FUNCTION_BLOCK fb_BusBrsEvent
VAR_INPUT
	 I_sID         			:STRING(10);     // Geräte-ID (z.B. '12345')
	 I_sInstID				:STRING(2) 	:=	'17';
	 I_sReceivedString		:STRING(255);	
	 I_bReset				:BOOL;
END_VAR
VAR_OUTPUT
	Q_lrBrs				:LREAL;
END_VAR
VAR	
	findStringTemp			:STRING;	(* Wird für TMP/ BRS/ RHD verwendet *)

	sBrs1					:STRING;
	sBrs2					:STRING;
	
END_VAR

findStringTemp	:= CONCAT(I_sID,'.');
findStringTemp	:= CONCAT(findStringTemp,'BRS');
findStringTemp	:= CONCAT(findStringTemp,'.');
findStringTemp	:= CONCAT(findStringTemp,I_sInstID);
findStringTemp	:= CONCAT(findStringTemp,'.');

IF I_bReset
THEN
	sBrs1 := '0';
ELSE
	IF FIND(I_sReceivedString,findStringTemp) >0 
	THEN
		sBrs1 :=MID(I_sReceivedString, (* LÄNGE*) 4, FIND(I_sReceivedString,'BRS.1.STATUS.')+ LEN('BRS.1.STATUS.'));
	END_IF
END_IF

Q_lrBrs :=	STRING_TO_LREAL(sBrs1);

END_FUNCTION_BLOCK

(* stored: Version 1.1.0.1, ProductVersion 3.1.4024.12
   POU fb_BusBrsEvent: Id {ce8deaea-2579-49df-9c5b-bc8e94fa1f43}, SpecialFunc None *)
